// Mitsubishi GX Works2 project: Ex2_done   PLC: FX3G

// global labels: Global1
VAR_GLOBAL
  locationSensor AT X001 : BOOL;
  Y_0 AT Y000 : BOOL;
  startMachine AT X010 : BOOL;
  EndZilufSensor AT X004 : BOOL;
  under15Temp AT X002 : BOOL;
  StopMachineZiluf AT X005 : BOOL;
  under30Temp AT X003 : BOOL;
  Y_5 AT Y005 : BOOL;
  ZilufOn AT Y004 : BOOL;
  x_7 AT X007 : BOOL;
  Y_7 AT Y007 : BOOL;
  startDaySwitch AT X007 : BOOL;
  choclateInput AT D1134 : REAL;
  ChoclateTank AT D1100 : REAL;
  creamTank AT D1102 : REAL;
  bisInput AT D1138 : REAL;
  bisTank AT D1104 : REAL;
  finishInput AT M1 : BOOL;
END_VAR
VAR_GLOBAL CONSTANT
  ChoclateRecipe : REAL := 240;
  ChoclateNeeded : REAL := 240;
  bisNeeded : REAL := 6;
END_VAR
VAR_GLOBAL
  notEnoughChoclate AT M2 : BOOL;
  notEnoughBis AT M3 : BOOL;
END_VAR
VAR_GLOBAL CONSTANT
  creamNeeded : REAL := 300;
END_VAR
VAR_GLOBAL
  notEnoughCreams AT M4 : BOOL;
  notEnoughMaterials AT M5 : BOOL;
  AnalogInput1 AT D8280 : INT;
END_VAR
VAR_GLOBAL CONSTANT
  const_w1 : INT := 1;
END_VAR
VAR_GLOBAL
  validInput1_greater AT M6 : BOOL;
END_VAR
VAR_GLOBAL CONSTANT
  const_w10 : INT := 10;
  const_w0 : INT;
END_VAR
VAR_GLOBAL
  validInput1_less AT M7 : BOOL;
  validInput1 AT M8 : BOOL;
  endOfDay AT M9 : BOOL;
  totalNumberofPacks AT D1106 : REAL;
END_VAR
VAR_GLOBAL CONSTANT
  multiplier : REAL := 0.6;
END_VAR
VAR_GLOBAL
  fictiveBlink AT M11 : BOOL;
END_VAR
VAR_GLOBAL CONSTANT
  blinkTime : INT := 5;
END_VAR
VAR_GLOBAL
  blink1Timer AT TC1 : BOOL;
  outputBlink1Timer AT TS1 : BOOL;
  fictiveLamp1 AT M12 : BOOL;
  blink2Timer AT TC2 : BOOL;
  outputBlink2Timer AT TS2 : BOOL;
  fictiveLamp2 AT M13 : BOOL;
  endDayTimer AT TC3 : BOOL;
END_VAR
VAR_GLOBAL CONSTANT
  dayBlinkTime : INT := 30;
END_VAR
VAR_GLOBAL
  outputEndDayTimer AT TS3 : BOOL;
  endDayBulb AT M15 : BOOL;
  zilufMachine AT D1108 : REAL;
  startDayBulb AT Y007 : BOOL;
  ActiveDay AT M16 : BOOL;
  creamInput AT D1136 : REAL;
  M_10 AT M10 : BOOL;
  Y_11 AT Y011 : BOOL;
  startCream AT X011 : BOOL;
END_VAR
VAR_GLOBAL CONSTANT
  CreamAmount : REAL := 300;
END_VAR
VAR_GLOBAL
  zilufTank AT D1110 : REAL;
END_VAR
VAR_GLOBAL CONSTANT
  transferAB : INT := 40;
END_VAR
VAR_GLOBAL
  TransferTimer AT TC4 : BOOL;
  blinking AT TC1 : BOOL;
  blinkingApply AT M17 : BOOL;
  StopBlinkingTransfer AT TS4 : BOOL;
  Y_01 AT Y001 : BOOL;
  normalDippingInput AT M20 : BOOL;
END_VAR
VAR_GLOBAL CONSTANT
  ChocklateAmount : REAL := 240;
  Double_ChoclateAmount : REAL := 240;
  Normal_ChoclateAmount : REAL := 120;
END_VAR
VAR_GLOBAL
  finishSampleDipping AT M21 : BOOL;
  DippingTimer AT D1114 : INT;
END_VAR
VAR_GLOBAL CONSTANT
  dippingTime : INT := 50;
END_VAR
VAR_GLOBAL
  DipTimer AT TC5 : BOOL;
END_VAR
VAR_GLOBAL CONSTANT
  dipTime : INT := 50;
END_VAR
VAR_GLOBAL
  endDipping AT TS5 : BOOL;
  y_3 AT Y003 : BOOL;
  dipAmount AT D1116 : REAL;
END_VAR
VAR_GLOBAL CONSTANT
  DoubleAmount : REAL := 240;
  NormalAmount : REAL := 120;
END_VAR
VAR_GLOBAL
  dippingTank AT D1118 : REAL;
END_VAR
VAR_GLOBAL CONSTANT
  const_w6 : INT := 6;
END_VAR
VAR_GLOBAL
  DoubleDippingInput AT M19 : BOOL;
  startDipping AT X006 : BOOL;
END_VAR
VAR_GLOBAL CONSTANT
  const_w5 : INT := 5;
  Nirmul : REAL := 120;
END_VAR
VAR_GLOBAL
  NormalInput1 AT D1122 : INT;
END_VAR
VAR_GLOBAL CONSTANT
  Nirmulnumber : INT := 388;
END_VAR
VAR_GLOBAL
  single_pack AT X000 : BOOL;
  Single_pack_counter AT CC1 : BOOL;
END_VAR
VAR_GLOBAL CONSTANT
  fiveKrambo : REAL := 5;
  five_krambo : INT := 5;
END_VAR
VAR_GLOBAL
  CS_1 AT CS1 : BOOL;
  Krambo_five_co AT CS1 : BOOL;
END_VAR
VAR_GLOBAL CONSTANT
  six_krambo : INT := 6;
END_VAR
VAR_GLOBAL
  six_pack_counter AT CC2 : BOOL;
  last_Krambo AT Y002 : BOOL;
  Total_counter AT CC3 : BOOL;
END_VAR
VAR_GLOBAL CONSTANT
  maxKrambo : INT := 1000;
END_VAR
VAR_GLOBAL
  kramboDailyAmount AT CN3 : INT;
END_VAR
VAR_GLOBAL CONSTANT
  Convertor_total_Krambo : INT := 10;
END_VAR
VAR_GLOBAL
  analogOutput AT D8282 : INT;
  counter_Restart AT CS2 : BOOL;
  Chek_X AT D1132 : INT;
  Check AT D1132 : INT;
END_VAR
VAR_GLOBAL CONSTANT
  Constantdiv : INT := 388;
END_VAR
VAR_GLOBAL
  endTransferTimer AT TS4 : BOOL;
  FinshTransferFlag AT M30 : BOOL;
  FinishTransferFlag AT M30 : BOOL;
  EndZilufStage AT M32 : BOOL;
  stage1_On AT M34 : BOOL;
  stage1_Off AT M35 : BOOL;
  stage4_Off AT M40 : BOOL;
  EndDipStage AT M37 : BOOL;
  stage3_Off AT M37 : BOOL;
  endCycle AT M42 : BOOL;
  MachineZilufOn AT M10 : BOOL;
  stage2_Off AT M36 : BOOL;
  TotalKrembos AT D1164 : INT;
  AnalogAnswer AT D1132 : INT;
  stage5_Off AT M90 : BOOL;
END_VAR

// task Task_01 (event TRUE, interval 0, priority 31): POU_01

PROGRAM POU_01
(* structured ladder/FBD written out as ST: instructions are called as NAME(EN, inputs, outputs); _pN, _eN, _tN stand for wires *)
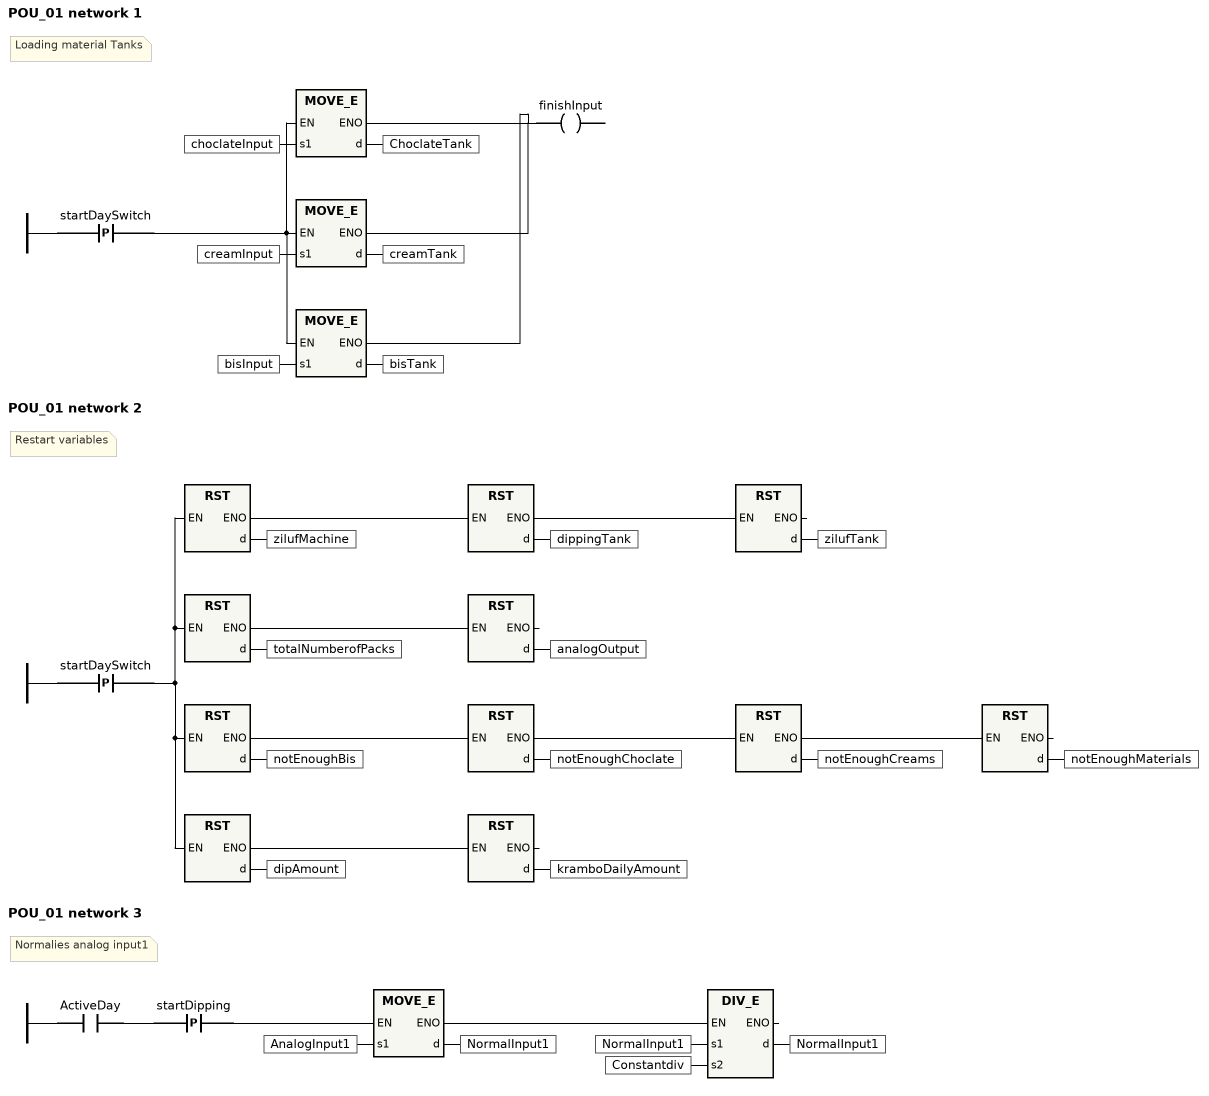
(* network 1 *)
(* Loading material Tanks *)
_p1 := LDP(TRUE, startDaySwitch);
_e2 := MOVE_E(_p1, choclateInput, ChoclateTank);
_e3 := MOVE_E(_p1, creamInput, creamTank);
_e4 := MOVE_E(_p1, bisInput, bisTank);
finishInput := _e2 OR _e3 OR _e4;
(* network 2 *)
(* Restart variables *)
_p1 := LDP(TRUE, startDaySwitch);
_e2 := RST(_p1, zilufMachine);
_e3 := RST(_e2, dippingTank);
RST(_e3, zilufTank);
_e4 := RST(_p1, totalNumberofPacks);
RST(_e4, analogOutput);
_e5 := RST(_p1, notEnoughBis);
_e6 := RST(_e5, notEnoughChoclate);
_e7 := RST(_e6, notEnoughCreams);
RST(_e7, notEnoughMaterials);
_e8 := RST(_p1, dipAmount);
RST(_e8, kramboDailyAmount);
(* network 3 *)
(* Normalies analog input1 *)
_e1 := MOVE_E(ActiveDay AND LDP(TRUE, startDipping), AnalogInput1, NormalInput1);
DIV_E(_e1, NormalInput1, Constantdiv, NormalInput1);
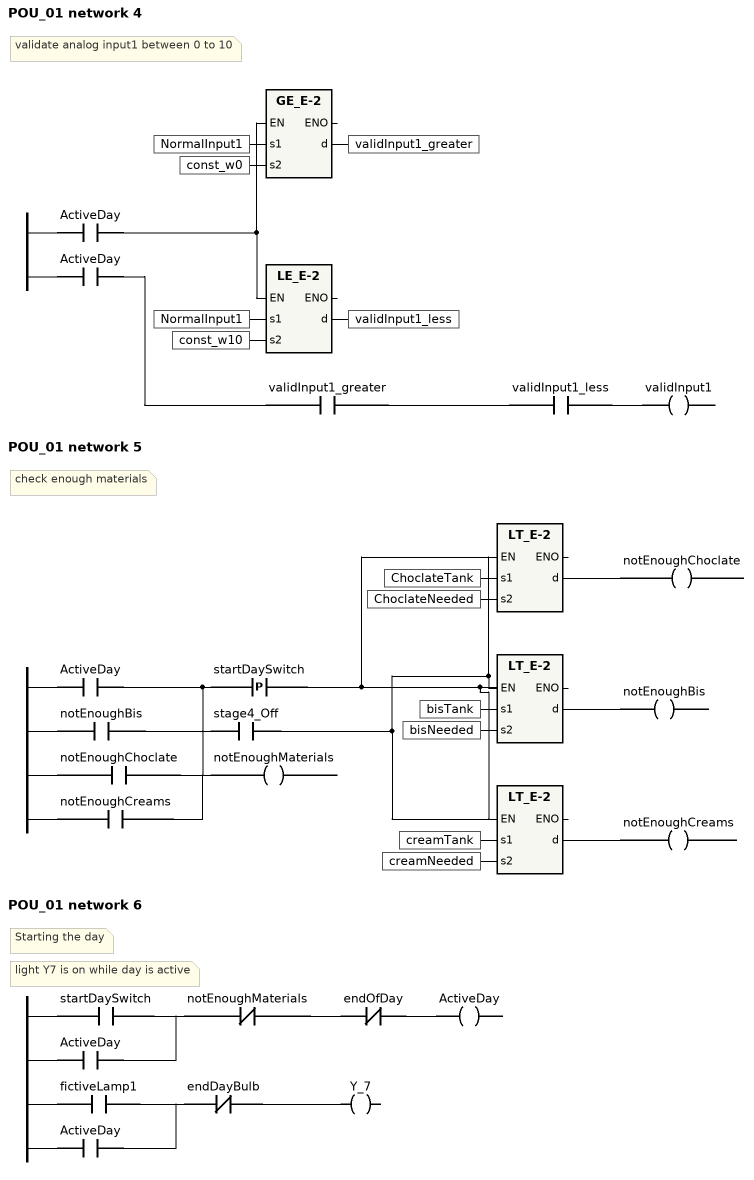
(* network 4 *)
(* validate analog input1 between 0 to 10 *)
GE_E(ActiveDay, NormalInput1, const_w0, validInput1_greater);
LE_E(ActiveDay, NormalInput1, const_w10, validInput1_less);
validInput1 := ActiveDay AND validInput1_greater AND validInput1_less;
(* network 5 *)
(* check enough materials *)
_p1 := (ActiveDay AND LDP(TRUE, startDaySwitch)) OR (ActiveDay AND stage4_Off);
LT_E(_p1, ChoclateTank, ChoclateNeeded, _t2);
notEnoughChoclate := _t2;
LT_E(_p1, bisTank, bisNeeded, _t3);
notEnoughBis := _t3;
LT_E(_p1, creamTank, creamNeeded, _t4);
notEnoughCreams := _t4;
notEnoughMaterials := notEnoughBis OR notEnoughChoclate OR notEnoughCreams;
(* network 6 *)
(* Starting the day *)
(* light Y7 is on while day is active *)
ActiveDay := ((startDaySwitch OR ActiveDay) AND NOT notEnoughMaterials) AND NOT endOfDay;
Y_7 := (fictiveLamp1 OR ActiveDay) AND NOT endDayBulb;
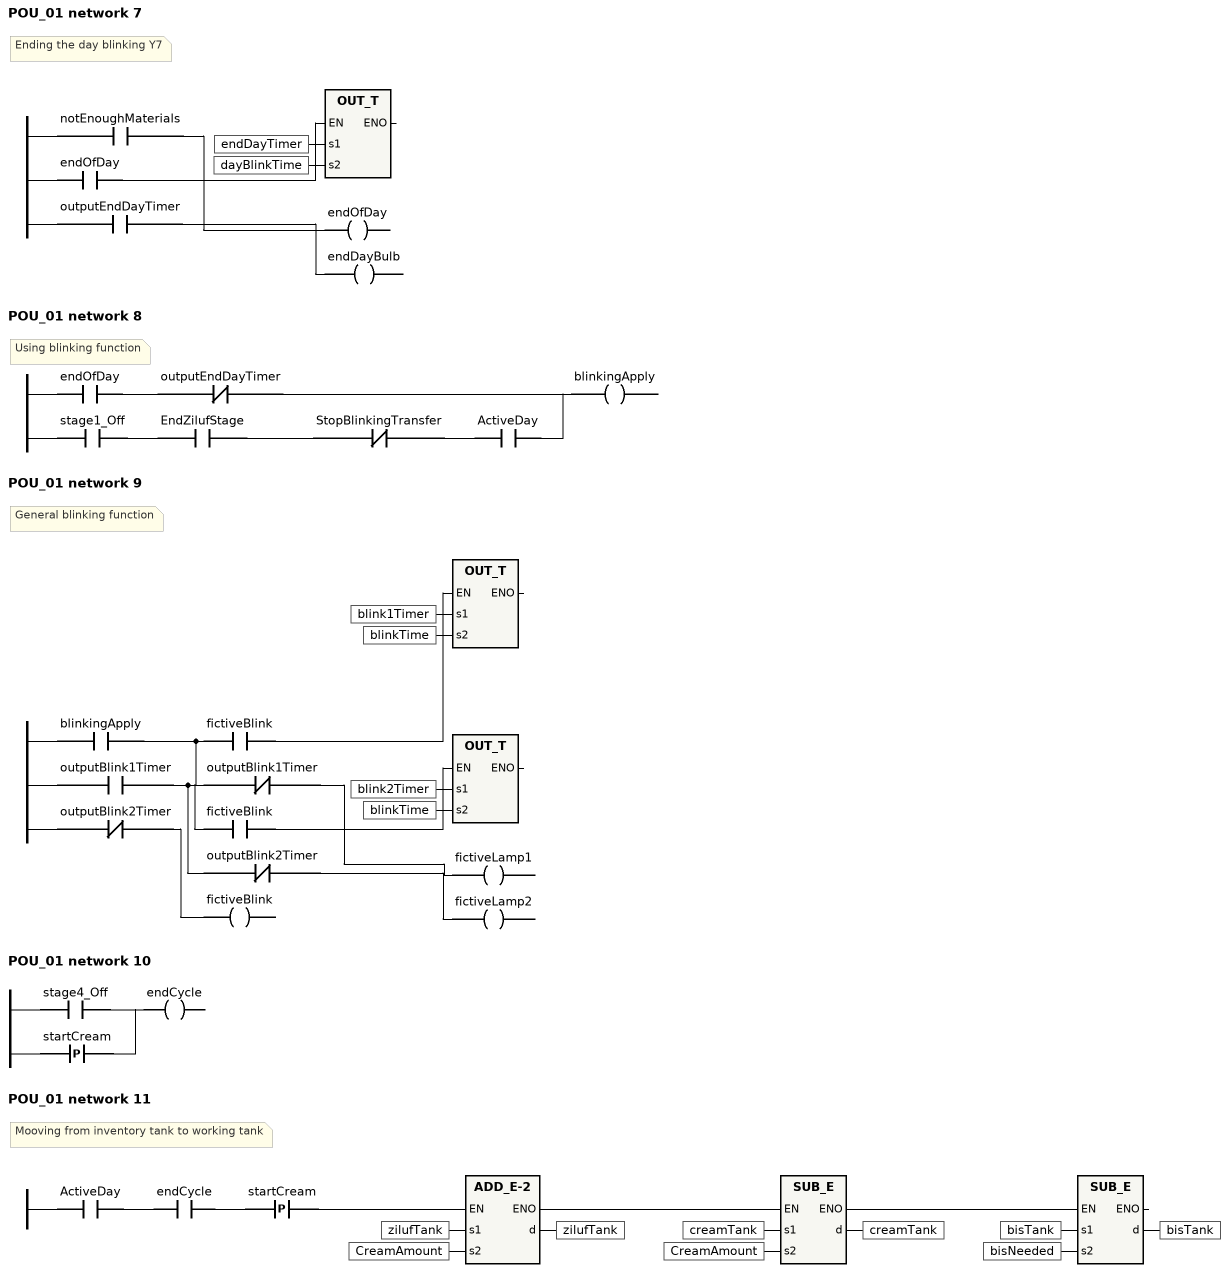
(* network 7 *)
(* Ending the day blinking Y7 *)
endOfDay := notEnoughMaterials;
OUT_T(endOfDay, endDayTimer, dayBlinkTime);
endDayBulb := outputEndDayTimer;
(* network 8 *)
(* Using blinking function *)
blinkingApply := (endOfDay AND NOT outputEndDayTimer) OR (stage1_Off AND EndZilufStage AND NOT StopBlinkingTransfer AND ActiveDay);
(* network 9 *)
(* General blinking function *)
OUT_T(blinkingApply AND fictiveBlink, blink1Timer, blinkTime);
fictiveLamp1 := blinkingApply AND NOT outputBlink1Timer;
OUT_T(outputBlink1Timer AND fictiveBlink, blink2Timer, blinkTime);
fictiveLamp2 := outputBlink1Timer AND NOT outputBlink2Timer;
fictiveBlink := NOT outputBlink2Timer;
(* network 10 *)
endCycle := stage4_Off OR LDP(TRUE, startCream);
(* network 11 *)
(* Mooving from inventory tank to working tank *)
_e1 := ADD_E(ActiveDay AND endCycle AND LDP(TRUE, startCream), zilufTank, CreamAmount, zilufTank);
_e2 := SUB_E(_e1, creamTank, CreamAmount, creamTank);
SUB_E(_e2, bisTank, bisNeeded, bisTank);
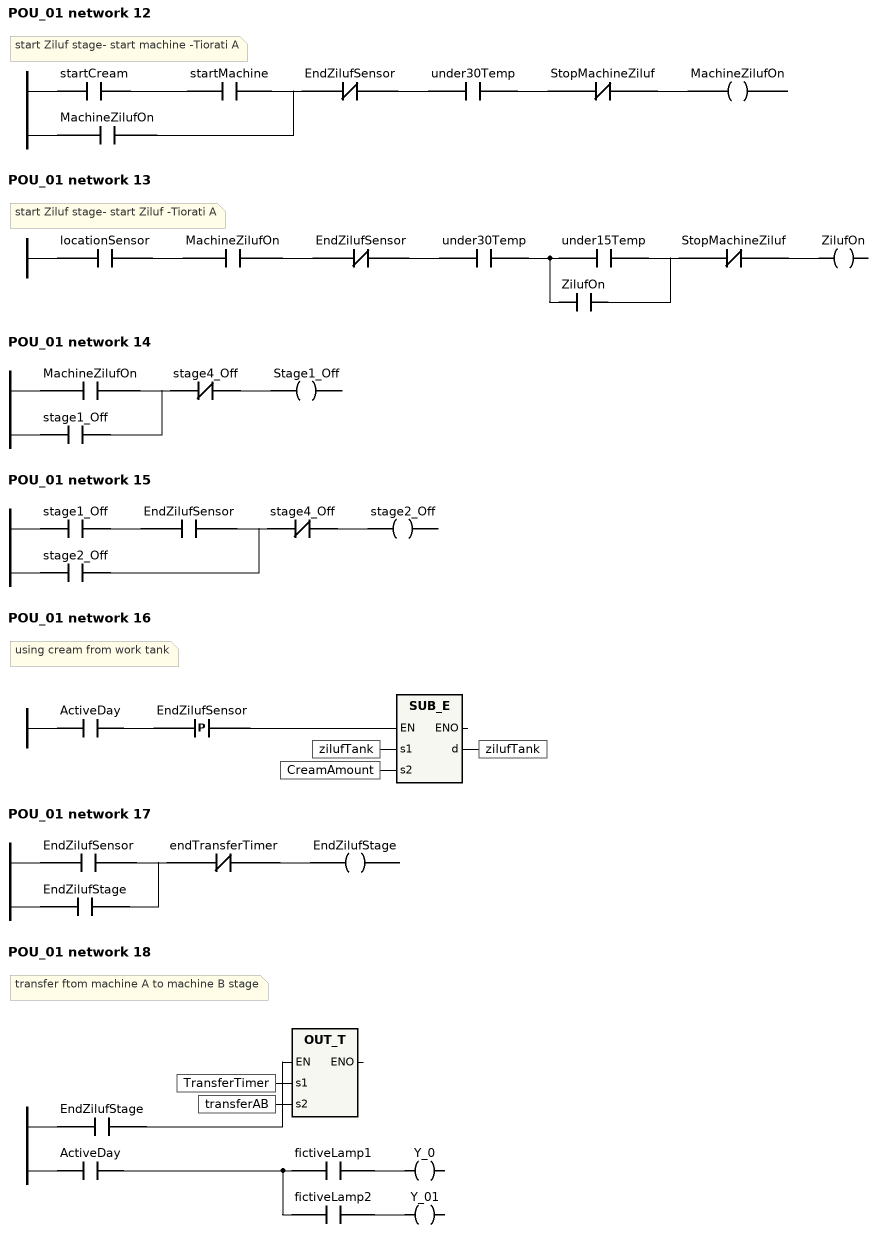
(* network 12 *)
(* start Ziluf stage- start machine -Tiorati A *)
MachineZilufOn := ((((startCream AND startMachine) OR MachineZilufOn) AND NOT EndZilufSensor) AND under30Temp) AND NOT StopMachineZiluf;
(* network 13 *)
(* start Ziluf stage- start Ziluf -Tiorati A *)
_p1 := locationSensor AND MachineZilufOn AND NOT EndZilufSensor AND under30Temp;
ZilufOn := ((_p1 AND under15Temp) OR (_p1 AND ZilufOn)) AND NOT StopMachineZiluf;
(* network 14 *)
Stage1_Off := (MachineZilufOn OR stage1_Off) AND NOT stage4_Off;
(* network 15 *)
stage2_Off := ((stage1_Off AND EndZilufSensor) OR stage2_Off) AND NOT stage4_Off;
(* network 16 *)
(* using cream from work tank *)
SUB_E(ActiveDay AND LDP(TRUE, EndZilufSensor), zilufTank, CreamAmount, zilufTank);
(* network 17 *)
EndZilufStage := (EndZilufSensor OR EndZilufStage) AND NOT endTransferTimer;
(* network 18 *)
(* transfer ftom machine A to machine B stage *)
OUT_T(EndZilufStage, TransferTimer, transferAB);
Y_0 := ActiveDay AND fictiveLamp1;
Y_01 := ActiveDay AND fictiveLamp2;
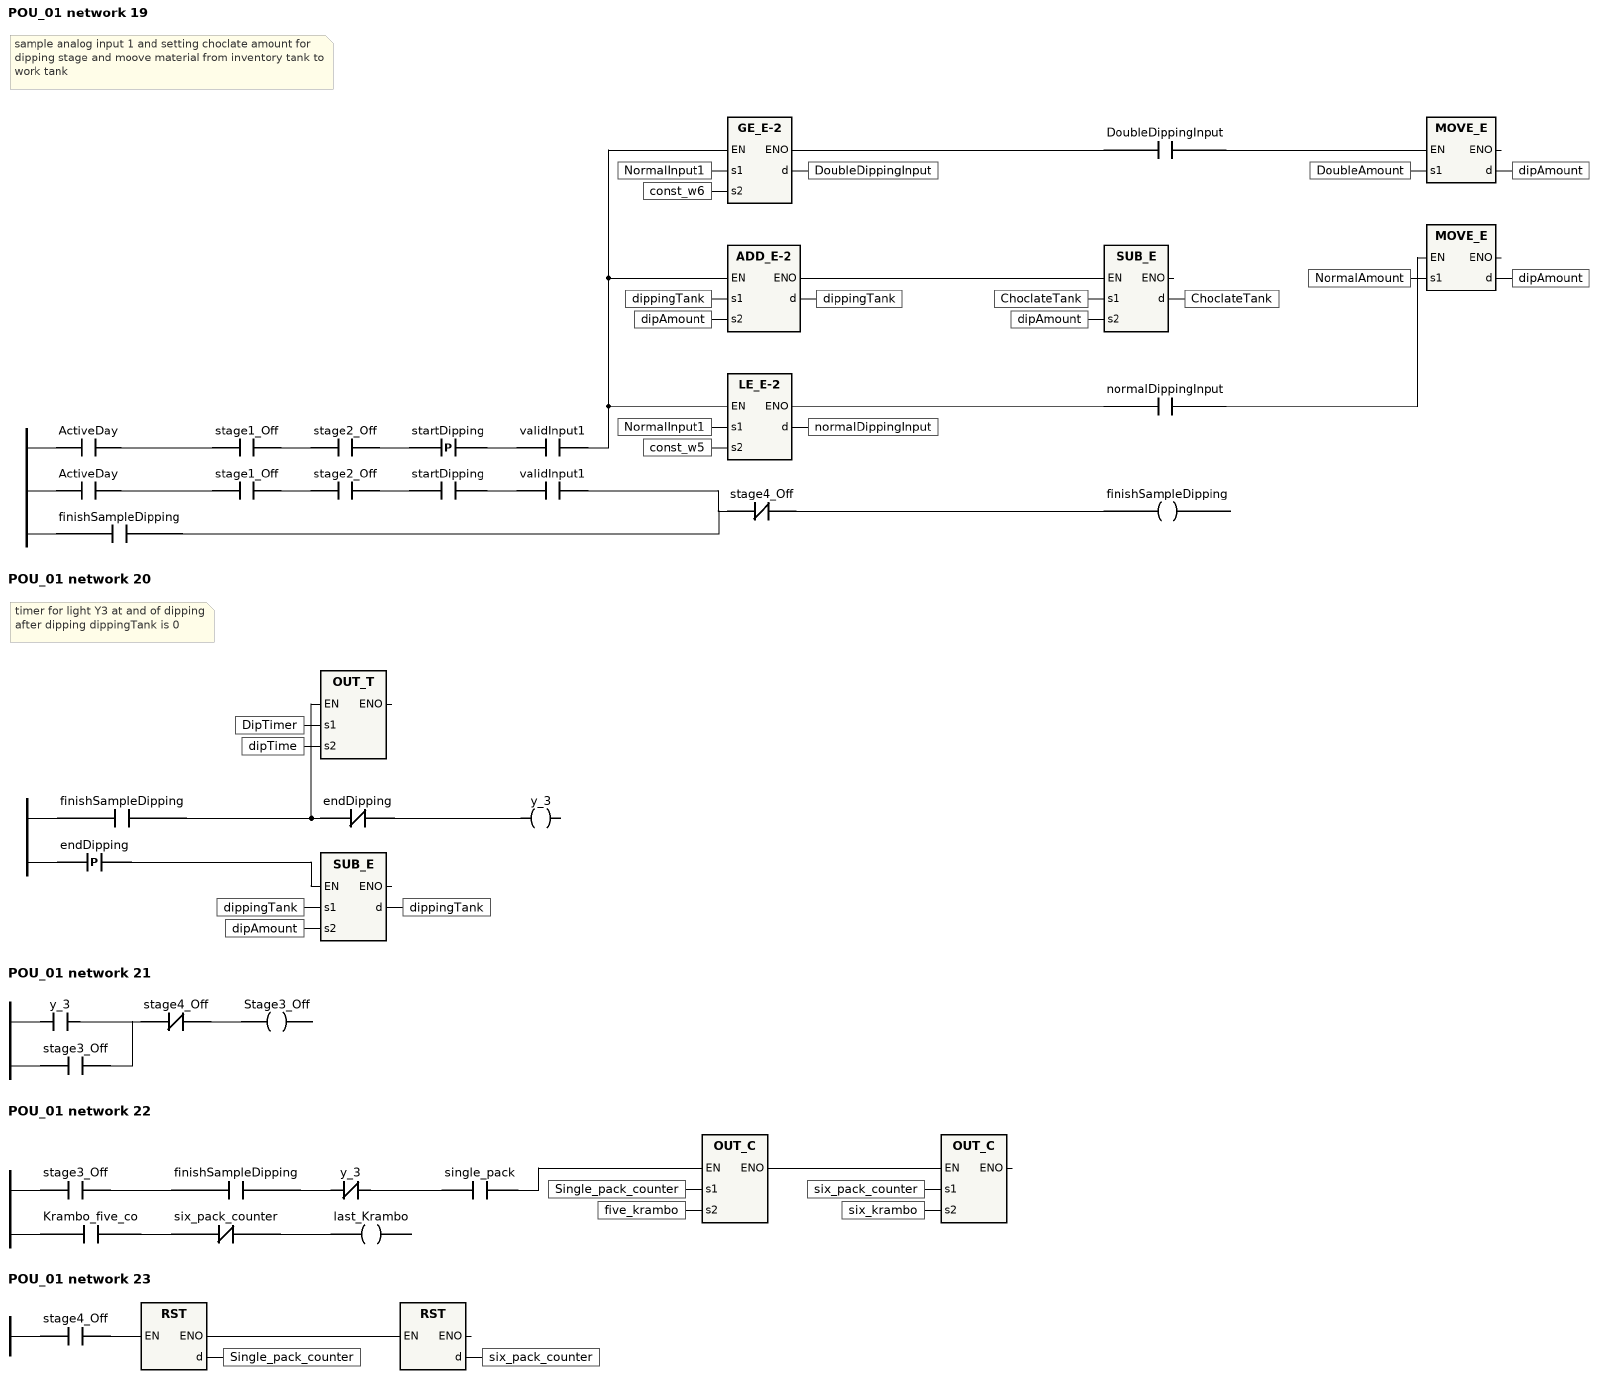
(* network 19 *)
(* sample analog input 1 and setting choclate amount for dipping stage and moove material from inventory tank to work tank *)
_p1 := ActiveDay AND stage1_Off AND stage2_Off AND LDP(TRUE, startDipping) AND validInput1;
_e2 := GE_E(_p1, NormalInput1, const_w6, DoubleDippingInput);
MOVE_E(_e2 AND DoubleDippingInput, DoubleAmount, dipAmount);
_e3 := LE_E(_p1, NormalInput1, const_w5, normalDippingInput);
MOVE_E(_e3 AND normalDippingInput, NormalAmount, dipAmount);
_e4 := ADD_E(_p1, dippingTank, dipAmount, dippingTank);
SUB_E(_e4, ChoclateTank, dipAmount, ChoclateTank);
finishSampleDipping := ((ActiveDay AND stage1_Off AND stage2_Off AND startDipping AND validInput1) OR finishSampleDipping) AND NOT stage4_Off;
(* network 20 *)
(* timer for light Y3 at and of dipping / after dipping dippingTank is 0 *)
OUT_T(finishSampleDipping, DipTimer, dipTime);
y_3 := finishSampleDipping AND NOT endDipping;
SUB_E(LDP(TRUE, endDipping), dippingTank, dipAmount, dippingTank);
(* network 21 *)
Stage3_Off := (y_3 OR stage3_Off) AND NOT stage4_Off;
(* network 22 *)
_e1 := OUT_C(stage3_Off AND finishSampleDipping AND NOT y_3 AND single_pack, Single_pack_counter, five_krambo);
OUT_C(_e1, six_pack_counter, six_krambo);
last_Krambo := Krambo_five_co AND NOT six_pack_counter;
(* network 23 *)
_e1 := RST(stage4_Off, Single_pack_counter);
RST(_e1, six_pack_counter);
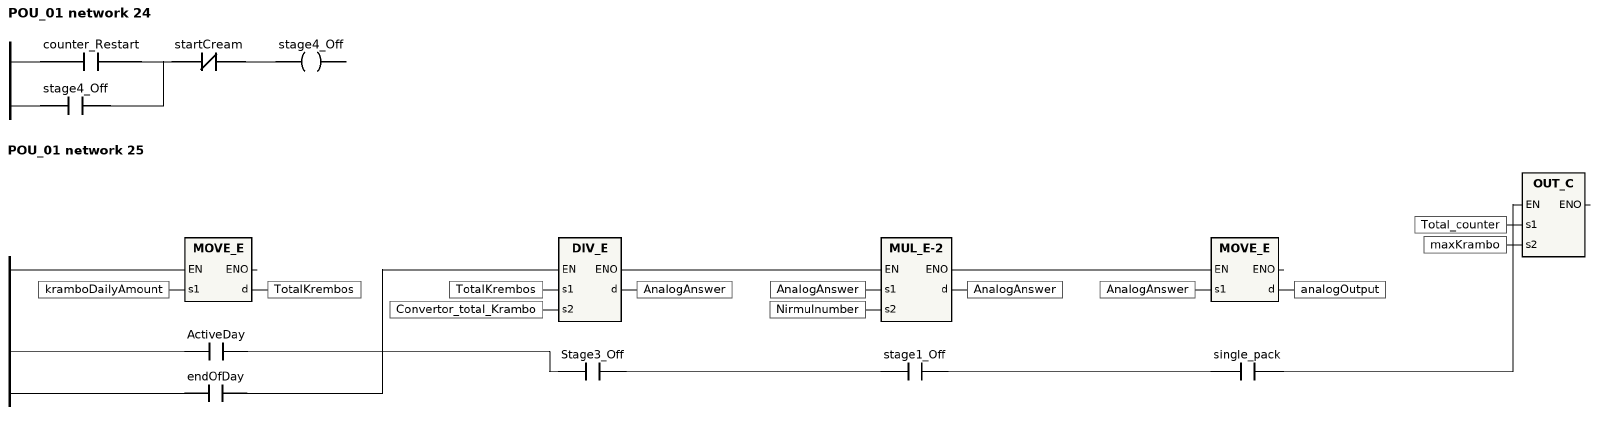
(* network 24 *)
stage4_Off := (counter_Restart OR stage4_Off) AND NOT startCream;
(* network 25 *)
OUT_C(ActiveDay AND Stage3_Off AND stage1_Off AND single_pack, Total_counter, maxKrambo);
MOVE_E(TRUE, kramboDailyAmount, TotalKrembos);
_e1 := DIV_E(endOfDay, TotalKrembos, Convertor_total_Krambo, AnalogAnswer);
_e2 := MUL_E(_e1, AnalogAnswer, Nirmulnumber, AnalogAnswer);
MOVE_E(_e2, AnalogAnswer, analogOutput);
END_PROGRAM
